(* IEC 61131-3 sources: com.logicals.lc3.webinar/usRTS_RPMControl_iSOC/src_FB_LIB_SAFE/Convert/USINT, 5 files *)

(* ---- wUSINT_TO_BYTE.iecst ---- *)
NAMESPACE logicals.web.standard
NAMESPACE convert

/*
 * Function block wrapper for IEC 61131-3 TO_BYTE<br>
 * IN =  input value (USINT)<br>
 * OUT = IN (BYTE)<br>
 */
FUNCTION_BLOCK wUSINT_TO_BYTE
	{ vNameAlignment:="center"; altName:="USINT_TO_BYTE"; bgColor:="DodgerBlue"; width:=140; hideIONames; }
	VAR_INPUT
		IN : USINT;
	END_VAR
	VAR_OUTPUT
		OUT: BYTE;
	END_VAR

	OUT := TO_BYTE(IN:=IN, ENO=>ENO);
END_FUNCTION_BLOCK

END_NAMESPACE
END_NAMESPACE

(* ---- wUSINT_TO_INT.iecst ---- *)
NAMESPACE logicals.web.standard
NAMESPACE convert

/*
 * Function block wrapper for IEC 61131-3 TO_INT<br>
 * IN =  input value (USINT)<br>
 * OUT = IN (INT)<br>
 */
FUNCTION_BLOCK wUSINT_TO_INT
	{ vNameAlignment:="center"; altName:="USINT_TO_INT"; bgColor:="LightPink"; width:=140; hideIONames; }
	VAR_INPUT
		IN : USINT;
	END_VAR
	VAR_OUTPUT
		OUT: INT;
	END_VAR

	OUT := TO_INT(IN:=IN, ENO=>ENO);
END_FUNCTION_BLOCK

END_NAMESPACE
END_NAMESPACE

(* ---- wUSINT_TO_UDINT.iecst ---- *)
NAMESPACE logicals.web.standard
NAMESPACE convert

/*
 * Function block wrapper for IEC 61131-3 TO_UDINT<br>
 * IN =  input value (USINT)<br>
 * OUT = IN (UDINT)<br>
 */
FUNCTION_BLOCK wUSINT_TO_UDINT
	{ vNameAlignment:="center"; altName:="USINT_TO_UDINT"; bgColor:="Plum"; width:=140; hideIONames; }
	VAR_INPUT
		IN : USINT;
	END_VAR
	VAR_OUTPUT
		OUT: UDINT;
	END_VAR

	OUT := TO_UDINT(IN:=IN, ENO=>ENO);
END_FUNCTION_BLOCK

END_NAMESPACE
END_NAMESPACE

(* ---- wUSINT_TO_UINT.iecst ---- *)
NAMESPACE logicals.web.standard
NAMESPACE convert

/*
 * Function block wrapper for IEC 61131-3 TO_UINT<br>
 * IN =  input value (USINT)<br>
 * OUT = IN (UINT)<br>
 */
FUNCTION_BLOCK wUSINT_TO_UINT
	{ vNameAlignment:="center"; altName:="USINT_TO_UINT"; bgColor:="Plum"; width:=140; hideIONames; }
	VAR_INPUT
		IN : USINT;
	END_VAR
	VAR_OUTPUT
		OUT: UINT;
	END_VAR

	OUT := TO_UINT(IN:=IN, ENO=>ENO);
END_FUNCTION_BLOCK

END_NAMESPACE
END_NAMESPACE

(* ---- wUSINT_TO_ULINT.iecst ---- *)
NAMESPACE logicals.web.standard
NAMESPACE convert

/*
 * Function block wrapper for IEC 61131-3 TO_ULINT<br>
 * IN =  input value (USINT)<br>
 * OUT = IN (ULINT)<br>
 */
FUNCTION_BLOCK wUSINT_TO_ULINT
	{ vNameAlignment:="center"; altName:="USINT_TO_ULINT"; bgColor:="Plum"; width:=140; hideIONames; }
	VAR_INPUT
		IN : USINT;
	END_VAR
	VAR_OUTPUT
		OUT: ULINT;
	END_VAR

	OUT := TO_ULINT(IN:=IN, ENO=>ENO);
END_FUNCTION_BLOCK

END_NAMESPACE
END_NAMESPACE
